// TIA Portal V16 export
// export: Created 2023-05-12T10:14:51.8633355Z, ExportSetting WithDefaults, DisplayName Totally Integrated Automation Portal, DisplayVersion V16 Update 3, DisplayName TIA Portal Version Control Interface, DisplayVersion V16 Update 2, DisplayName TIA Portal Openness, DisplayVersion V16 Update 3, DisplayName SINAMICS Startdrive Advanced, DisplayVersion V16, DisplayName SINAMICS Startdrive G130, G150, S120, S150, SINAMICS MV, S210, DisplayVersion V16, DisplayName SINAMICS Startdrive G110M, G120, G120C, G120D, G120P, DisplayVersion V16, DisplayName STEP 7 Professional, DisplayVersion V16 Update 3, DisplayName STEP 7 Safety, DisplayVersion V16, DisplayName WinCC Advanced, DisplayVersion V16 Update 3
FUNCTION "CAUDALES" : Void   // FC5, STL
{ S7_Optimized_Access := 'FALSE' }
VERSION : 0.1
// prueba
// stored: AutoNumber false, ParameterPassing false, UDAEnableTagReadback false
BEGIN

NETWORK
TITLE = BOMBA BC-14. ENTRADA PRODUCTO PASTER

      CALL  SCALE
      ( IN      := "Tag_83":P,
        HI_LIM  := 10000.0,
        LO_LIM  := -5.5,
        BIPOLAR := FALSE,
        RET_VAL := "Tag_6",
        OUT     := "CAUDAL PASTER 4000".CAUDAL_REAL
      );


      CALL  "CONTROL CAUDAL", "CAUDAL PASTER 4000"
      ( SET_POINT_CAUDAL  := ,
        HIST_ALTA_CAUDAL  := ,
        HIST_BAJA_CAUDAL  := ,
        ALARM_ALTA_CAUDAL := ,
        ALARM_BAJA_CAUDAL := ,
        CAUDAL_REAL       := ,
        ALARM_CAUDAL_ALTA := ,
        ALARM_CAUDAL_BAJA := ,
        CAUDAL_OK         := ,
        SP_CAUDAL_MANUAL  := 
      );

NETWORK
TITLE = CAUDAL LINEA GELATINA/ DENSIDAD/ PRUEBAS

      CALL  SCALE
      ( IN      := "Tag_84":P,
        HI_LIM  := 6000.0,
        LO_LIM  := 0.0,
        BIPOLAR := FALSE,
        RET_VAL := "Tag_6",
        OUT     := "CAUDAL MASICO GELATINA".CAUDAL_REAL
      );


      CALL  "CONTROL CAUDAL", "CAUDAL MASICO GELATINA"
      ( SET_POINT_CAUDAL  := ,
        HIST_ALTA_CAUDAL  := ,
        HIST_BAJA_CAUDAL  := ,
        ALARM_ALTA_CAUDAL := ,
        ALARM_BAJA_CAUDAL := 250.0,  // 5.000000e+002 //9.000000e+002
        CAUDAL_REAL       := ,
        ALARM_CAUDAL_ALTA := ,
        ALARM_CAUDAL_BAJA := ,
        CAUDAL_OK         := ,
        SP_CAUDAL_MANUAL  := 
      );

NETWORK
TITLE = CAUDAL LINEA DOSIFICADO ACIDO EN GELATINA
// OJO LA ENTRADA ANALOGICA UTILIZADA ESTA AHORA CON LA SEÑAL DE RESERVA DEL MASICO
//  la PEW510

//     CALL  "SCALE"
//       IN     :=
//       HI_LIM :=3.000000e+001
//       LO_LIM :=0.000000e+000
//       BIPOLAR:=FALSE
//       RET_VAL:=MW100
//       OUT    :="CAUDAL ACIDO".CAUDAL_REAL


//      CALL  "CONTROL CAUDAL" , "CAUDAL ACIDO"
//       SET_POINT_CAUDAL :=
//       HIST_ALTA_CAUDAL :=
//       HIST_BAJA_CAUDAL :=
//       ALARM_ALTA_CAUDAL:=
//       ALARM_BAJA_CAUDAL:=
//       CAUDAL_REAL      :=
//       ALARM_CAUDAL_ALTA:=
//       ALARM_CAUDAL_BAJA:=
//       CAUDAL_OK        :=
//       SP_CAUDAL_MANUAL :=

NETWORK
TITLE = 

//      U     E    152.5
//      ZV    Z     50


NETWORK
TITLE = CAUDAL LINEA PASTERIZADOR 2500

      CALL  SCALE
      ( IN      := "Tag_85":P,
        HI_LIM  := 5000.0,
        LO_LIM  := -5.7,
        BIPOLAR := FALSE,
        RET_VAL := "Tag_6",
        OUT     := "CAUDAL PASTER 2500".CAUDAL_REAL
      );


      CALL  "CONTROL CAUDAL", "CAUDAL PASTER 2500"
      ( SET_POINT_CAUDAL  := ,
        HIST_ALTA_CAUDAL  := ,
        HIST_BAJA_CAUDAL  := ,
        ALARM_ALTA_CAUDAL := ,
        ALARM_BAJA_CAUDAL := ,
        CAUDAL_REAL       := ,
        ALARM_CAUDAL_ALTA := ,
        ALARM_CAUDAL_BAJA := ,
        CAUDAL_OK         := ,
        SP_CAUDAL_MANUAL  := 
      );
END_FUNCTION
